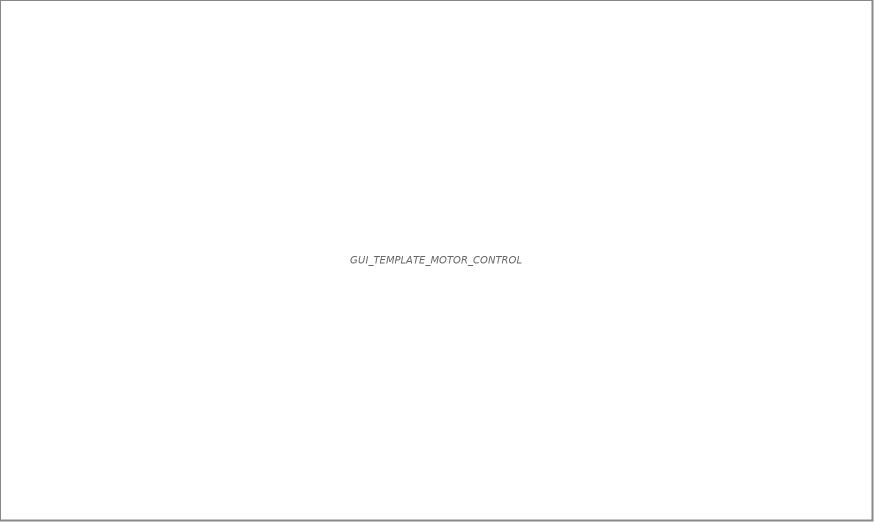
VISUALIZATION GUI_Motor002_Ctrl  // 874x522
    Frame (0,0 872x520)
        shows GUI_TEMPLATE_MOTOR_CONTROL(m_Instance := MAIN.Motor002)
END_VISUALIZATION

(* stored: Version 1.1.0.1, ProductVersion 3.1.4024.3
   Visu GUI_Motor002_Ctrl: Id {420d8475-112d-44c3-9925-bc7889ecee26} *)
